(* PLC project  *)

PROGRAM P

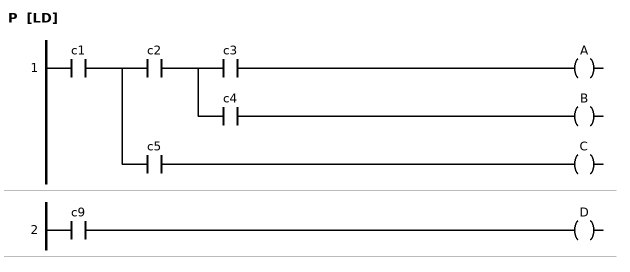
(* LD diagram, written out as Structured Text *)
A := c1 AND c2 AND c3;
B := c1 AND c2 AND c4;
C := c1 AND c5;
D := c9;
END_PROGRAM
